// TIA Portal V16 export
// export: Created 2025-10-07T21:39:07.5159654Z, ExportSetting WithDefaults, DisplayName Totally Integrated Automation Portal, DisplayVersion V16, DisplayName TIA Portal Version Control Interface, DisplayVersion V16, DisplayName TIA Portal Openness, DisplayVersion V16, DisplayName STEP 7 Professional, DisplayVersion V16, DisplayName STEP 7 Safety, DisplayVersion V16, DisplayName WinCC Advanced, DisplayVersion V16
FUNCTION "5 - Prog. 3" : Void   // FC3, LAD
TITLE = System Program 3
VERSION : 0.1
// stored: AutoNumber true, IsIECCheckEnabled false, UDAEnableTagReadback false
   VAR_TEMP
      BlowOffTimer : Bool;
      Democoil : Bool;
      StartBlowOff : Bool;
      Pos2_Done : Bool;
      BlowOff_Activated : Bool;
      Retourband_Delayed : Bool;
      AandrukCilindersOut : Bool;
      Move2Busy : Bool;
      ProductBehindWals : Bool;
      SR_Move2 : Bool;
      Move1Busy : Bool;
   END_VAR
   VAR_TEMP   // added for the SCL form of the ladder/FBD networks
      _w1 : Bool;
   END_VAR
BEGIN

REGION Network 1: Close 1 Magazine Hole (cilinder)
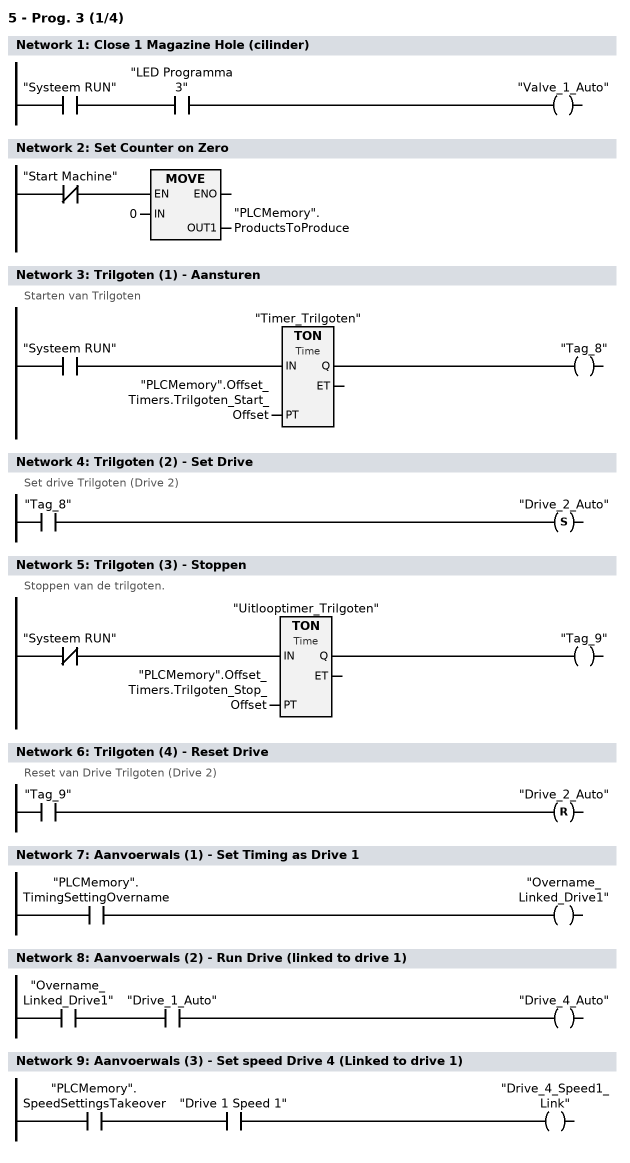
   RUNG wire#powerrail
      Contact( "Systeem RUN" )
      Contact( "LED Programma 3" )
      Coil( "Valve_1_Auto" )
   END_RUNG
   // the same network as SCL:
   "Valve_1_Auto" := "Systeem RUN" AND "LED Programma 3";
END_REGION

REGION Network 2: Set Counter on Zero
   RUNG wire#powerrail
      I_Contact( "Start Machine" )
      { S7_GenerateENO := "TRUE" } Move(in := 0, out1 => "PLCMemory".ProductsToProduce)
   END_RUNG
   // the same network as SCL:
   IF NOT "Start Machine" THEN "PLCMemory".ProductsToProduce := 0; END_IF;
END_REGION

REGION Network 3: Trilgoten (1) - Aansturen
   // Starten van Trilgoten
   RUNG wire#powerrail
      Contact( "Systeem RUN" )
      { S7_Templates := "time_type := Time" } "Timer_Trilgoten".TON(pt := "PLCMemory".Offset_Timers.Trilgoten_Start_Offset, et =>)
      Coil( "Tag_8" )
   END_RUNG
   // the same network as SCL:
   "Timer_Trilgoten".TON(IN := "Systeem RUN", PT := "PLCMemory".Offset_Timers.Trilgoten_Start_Offset);
   "Tag_8" := "Timer_Trilgoten".Q;
END_REGION

REGION Network 4: Trilgoten (2) - Set Drive
   // Set drive Trilgoten (Drive 2)
   RUNG wire#powerrail
      Contact( "Tag_8" )
      S_Coil( "Drive_2_Auto" )
   END_RUNG
   // the same network as SCL:
   IF "Tag_8" THEN "Drive_2_Auto" := TRUE; END_IF;
END_REGION

REGION Network 5: Trilgoten (3) - Stoppen
   // Stoppen van de trilgoten.
   RUNG wire#powerrail
      I_Contact( "Systeem RUN" )
      { S7_Templates := "time_type := Time" } "Uitlooptimer_Trilgoten".TON(pt := "PLCMemory".Offset_Timers.Trilgoten_Stop_Offset, et =>)
      Coil( "Tag_9" )
   END_RUNG
   // the same network as SCL:
   "Uitlooptimer_Trilgoten".TON(IN := NOT "Systeem RUN", PT := "PLCMemory".Offset_Timers.Trilgoten_Stop_Offset);
   "Tag_9" := "Uitlooptimer_Trilgoten".Q;
END_REGION

REGION Network 6: Trilgoten (4) - Reset Drive
   // Reset van Drive Trilgoten (Drive 2)
   RUNG wire#powerrail
      Contact( "Tag_9" )
      R_Coil( "Drive_2_Auto" )
   END_RUNG
   // the same network as SCL:
   IF "Tag_9" THEN "Drive_2_Auto" := FALSE; END_IF;
END_REGION

REGION Network 7: Aanvoerwals (1) - Set Timing as Drive 1
   RUNG wire#powerrail
      Contact( "PLCMemory".TimingSettingOvername )
      Coil( "Overname_Linked_Drive1" )
   END_RUNG
   // the same network as SCL:
   "Overname_Linked_Drive1" := "PLCMemory".TimingSettingOvername;
END_REGION

REGION Network 8: Aanvoerwals (2) - Run Drive (linked to drive 1)
   RUNG wire#powerrail
      Contact( "Overname_Linked_Drive1" )
      Contact( "Drive_1_Auto" )
      Coil( "Drive_4_Auto" )
   END_RUNG
   // the same network as SCL:
   "Drive_4_Auto" := "Overname_Linked_Drive1" AND "Drive_1_Auto";
END_REGION

REGION Network 9: Aanvoerwals (3) - Set speed Drive 4 (Linked to drive 1)
   RUNG wire#powerrail
      Contact( "PLCMemory".SpeedSettingsTakeover )
      Contact( "Drive 1 Speed 1" )
      Coil( "Drive_4_Speed1_Link" )
   END_RUNG
   // the same network as SCL:
   "Drive_4_Speed1_Link" := "PLCMemory".SpeedSettingsTakeover AND "Drive 1 Speed 1";
END_REGION

REGION Network 10: Aanvoerwals (4) - Set alternative Speed 1
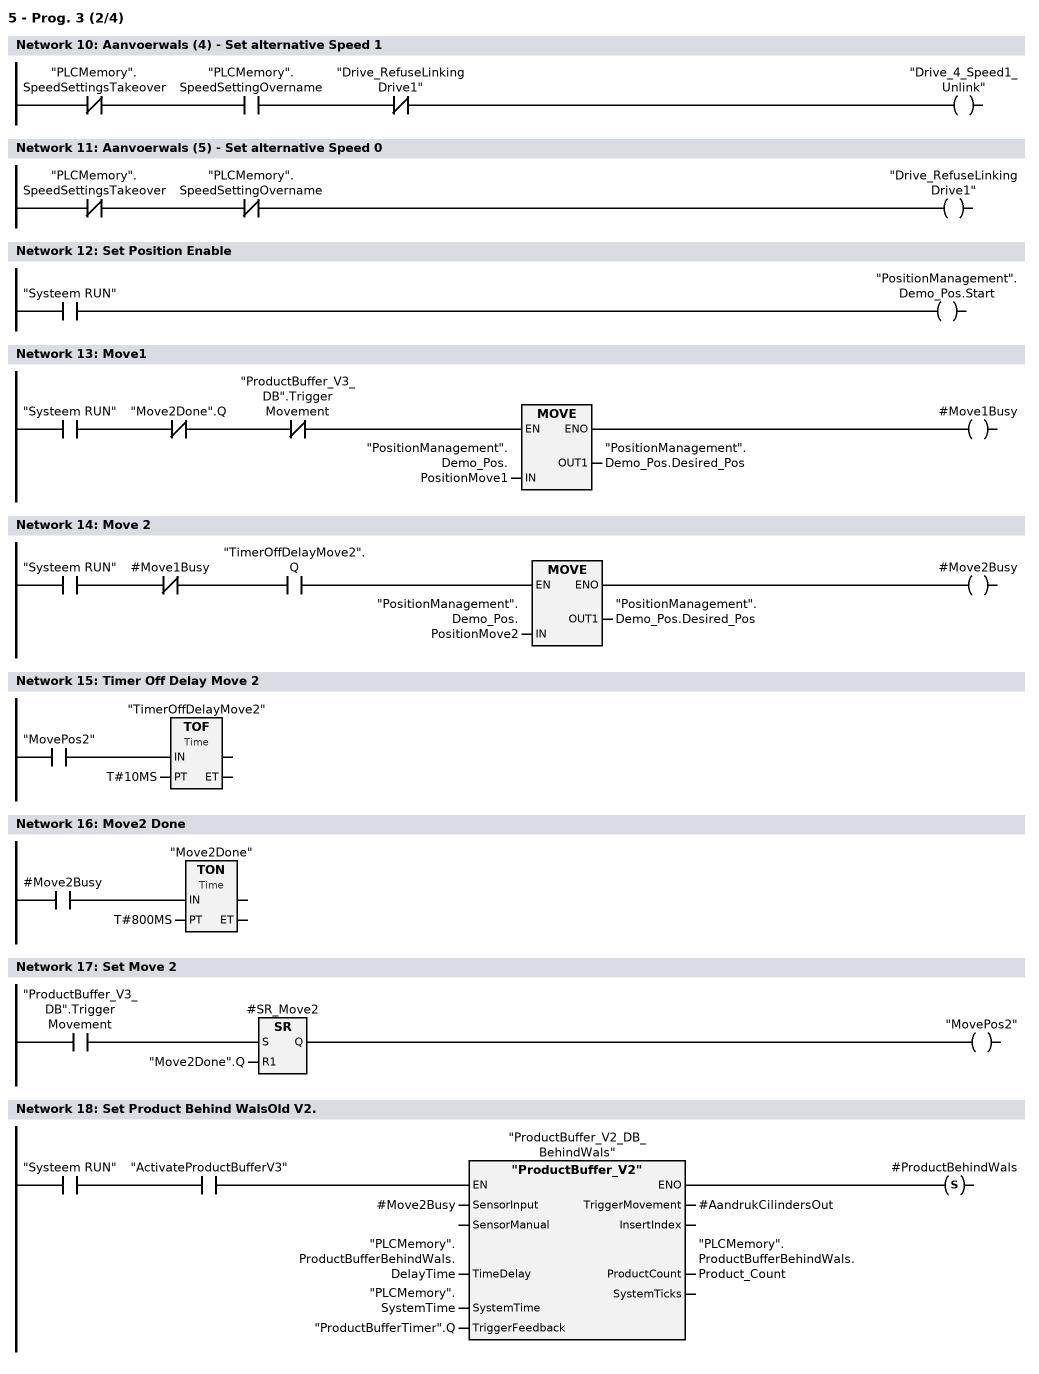
   RUNG wire#powerrail
      I_Contact( "PLCMemory".SpeedSettingsTakeover )
      Contact( "PLCMemory".SpeedSettingOvername )
      I_Contact( "Drive_RefuseLinkingDrive1" )
      Coil( "Drive_4_Speed1_Unlink" )
   END_RUNG
   // the same network as SCL:
   "Drive_4_Speed1_Unlink" := NOT "PLCMemory".SpeedSettingsTakeover AND "PLCMemory".SpeedSettingOvername AND NOT "Drive_RefuseLinkingDrive1";
END_REGION

REGION Network 11: Aanvoerwals (5) - Set alternative Speed 0
   RUNG wire#powerrail
      I_Contact( "PLCMemory".SpeedSettingsTakeover )
      I_Contact( "PLCMemory".SpeedSettingOvername )
      Coil( "Drive_RefuseLinkingDrive1" )
   END_RUNG
   // the same network as SCL:
   "Drive_RefuseLinkingDrive1" := NOT "PLCMemory".SpeedSettingsTakeover AND NOT "PLCMemory".SpeedSettingOvername;
END_REGION

REGION Network 12: Set Position Enable
   RUNG wire#powerrail
      Contact( "Systeem RUN" )
      Coil( "PositionManagement".Demo_Pos.Start )
   END_RUNG
   // the same network as SCL:
   "PositionManagement".Demo_Pos.Start := "Systeem RUN";
END_REGION

REGION Network 13: Move1
   RUNG wire#powerrail
      Contact( "Systeem RUN" )
      I_Contact( "Move2Done".Q )
      I_Contact( "ProductBuffer_V3_DB".TriggerMovement )
      { S7_GenerateENO := "TRUE" } Move(in := "PositionManagement".Demo_Pos.PositionMove1, out1 => "PositionManagement".Demo_Pos.Desired_Pos)
      Coil( #Move1Busy )
   END_RUNG
   // the same network as SCL:
   // ENO of a box is taken as its EN; it also drops when the box reports an error
   #_w1 := "Systeem RUN" AND NOT "Move2Done".Q AND NOT "ProductBuffer_V3_DB".TriggerMovement;
   IF #_w1 THEN
       "PositionManagement".Demo_Pos.Desired_Pos := "PositionManagement".Demo_Pos.PositionMove1;
   END_IF;
   #Move1Busy := #_w1;
END_REGION

REGION Network 14: Move 2
   RUNG wire#powerrail
      Contact( "Systeem RUN" )
      I_Contact( #Move1Busy )
      Contact( "TimerOffDelayMove2".Q )
      { S7_GenerateENO := "TRUE" } Move(in := "PositionManagement".Demo_Pos.PositionMove2, out1 => "PositionManagement".Demo_Pos.Desired_Pos)
      Coil( #Move2Busy )
   END_RUNG
   // the same network as SCL:
   // ENO of a box is taken as its EN; it also drops when the box reports an error
   #_w1 := "Systeem RUN" AND NOT #Move1Busy AND "TimerOffDelayMove2".Q;
   IF #_w1 THEN
       "PositionManagement".Demo_Pos.Desired_Pos := "PositionManagement".Demo_Pos.PositionMove2;
   END_IF;
   #Move2Busy := #_w1;
END_REGION

REGION Network 15: Timer Off Delay Move 2
   RUNG wire#powerrail
      Contact( "MovePos2" )
      { S7_Templates := "time_type := Time" } "TimerOffDelayMove2".TOF(pt := T#10MS, et =>)
   END_RUNG
   // the same network as SCL:
   "TimerOffDelayMove2".TOF(IN := "MovePos2", PT := T#10MS);
END_REGION

REGION Network 16: Move2 Done
   RUNG wire#powerrail
      Contact( #Move2Busy )
      { S7_Templates := "time_type := Time" } "Move2Done".TON(pt := T#800MS, et =>)
   END_RUNG
   // the same network as SCL:
   "Move2Done".TON(IN := #Move2Busy, PT := T#800MS);
END_REGION

REGION Network 17: Set Move 2
   RUNG wire#powerrail
      Contact( "ProductBuffer_V3_DB".TriggerMovement )
      S_SR(operand := #SR_Move2, r1 := "Move2Done".Q)
      Coil( "MovePos2" )
   END_RUNG
   // the same network as SCL:
   IF "ProductBuffer_V3_DB".TriggerMovement THEN
       #SR_Move2 := TRUE;   // SR flip-flop
   END_IF;
   IF "Move2Done".Q THEN #SR_Move2 := FALSE; END_IF;
   "MovePos2" := #SR_Move2;
END_REGION

REGION Network 18: Set Product Behind WalsOld V2.
   RUNG wire#powerrail
      Contact( "Systeem RUN" )
      Contact( "ActivateProductBufferV3" )
      "ProductBuffer_V2_DB_BehindWals"(SensorInput := #Move2Busy, SensorManual :=, TimeDelay := "PLCMemory".ProductBufferBehindWals.DelayTime, SystemTime := "PLCMemory".SystemTime, TriggerFeedback := "ProductBufferTimer".Q, TriggerMovement => #AandrukCilindersOut, InsertIndex =>, ProductCount => "PLCMemory".ProductBufferBehindWals.Product_Count, SystemTicks =>)
      S_Coil( #ProductBehindWals )
   END_RUNG
   // the same network as SCL:
   "ProductBuffer_V2_DB_BehindWals"(EN := "Systeem RUN" AND "ActivateProductBufferV3",   // "ProductBuffer_V2"
                           SensorInput := #Move2Busy,
                           TimeDelay := "PLCMemory".ProductBufferBehindWals.DelayTime,
                           SystemTime := "PLCMemory".SystemTime,
                           TriggerFeedback := "ProductBufferTimer".Q,
                           TriggerMovement => #AandrukCilindersOut,
                           ProductCount => "PLCMemory".ProductBufferBehindWals.Product_Count,
                           ENO => #_w1);
   IF #_w1 THEN #ProductBehindWals := TRUE; END_IF;
END_REGION

REGION Network 19: PorductBuffer Behind Wals V3
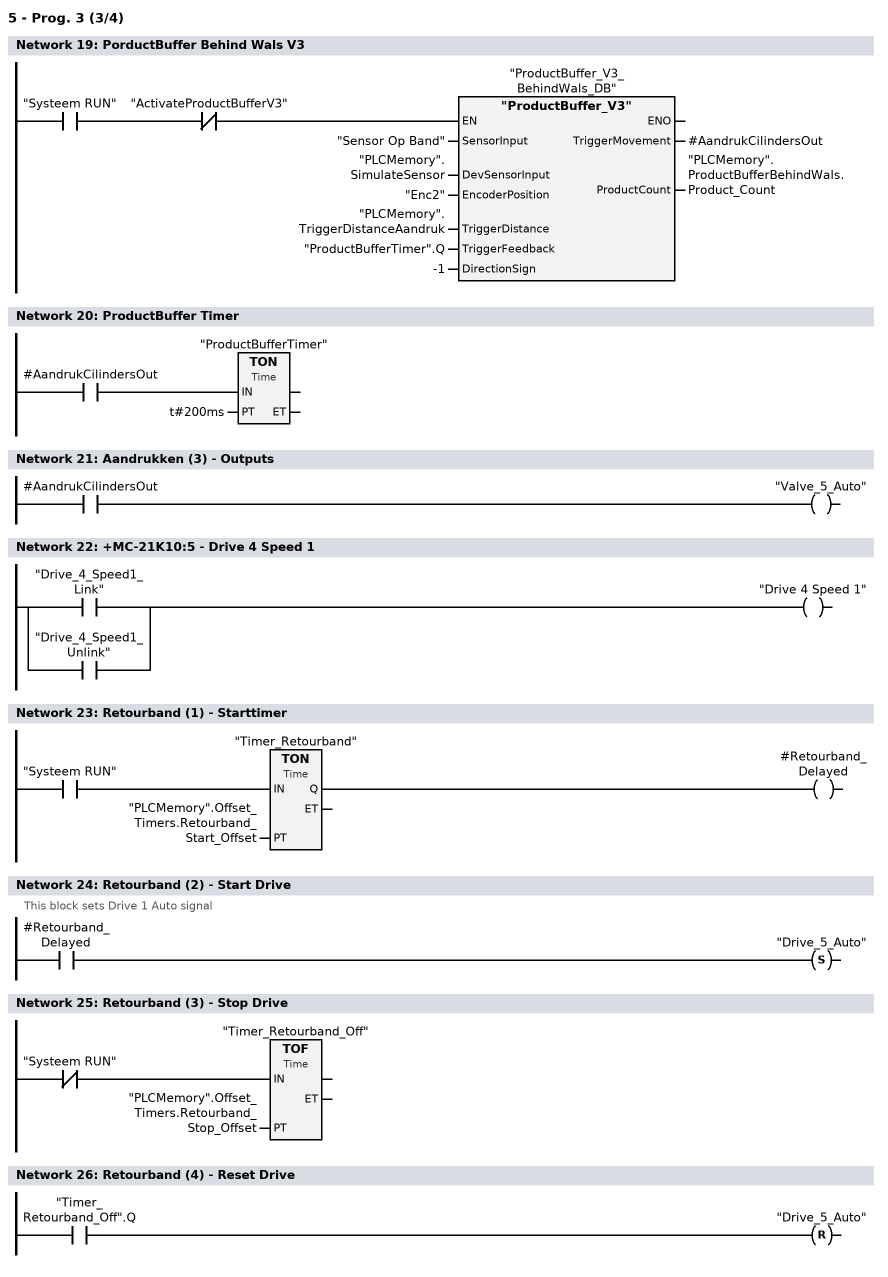
   RUNG wire#powerrail
      Contact( "Systeem RUN" )
      I_Contact( "ActivateProductBufferV3" )
      "ProductBuffer_V3_BehindWals_DB"(SensorInput := "Sensor Op Band", DevSensorInput := "PLCMemory".SimulateSensor, EncoderPosition := "Enc2", TriggerDistance := "PLCMemory".TriggerDistanceAandruk, TriggerFeedback := "ProductBufferTimer".Q, DirectionSign := -1, TriggerMovement => #AandrukCilindersOut, ProductCount => "PLCMemory".ProductBufferBehindWals.Product_Count)
   END_RUNG
   // the same network as SCL:
   IF "Systeem RUN" AND NOT "ActivateProductBufferV3" THEN
       "ProductBuffer_V3_BehindWals_DB"(SensorInput := "Sensor Op Band",   // "ProductBuffer_V3"
                               DevSensorInput := "PLCMemory".SimulateSensor,
                               EncoderPosition := "Enc2",
                               TriggerDistance := "PLCMemory".TriggerDistanceAandruk,
                               TriggerFeedback := "ProductBufferTimer".Q,
                               DirectionSign := -1,
                               TriggerMovement => #AandrukCilindersOut,
                               ProductCount => "PLCMemory".ProductBufferBehindWals.Product_Count);
   END_IF;
END_REGION

REGION Network 20: ProductBuffer Timer
   RUNG wire#powerrail
      Contact( #AandrukCilindersOut )
      { S7_Templates := "time_type := Time" } "ProductBufferTimer".TON(pt := t#200ms, et =>)
   END_RUNG
   // the same network as SCL:
   "ProductBufferTimer".TON(IN := #AandrukCilindersOut, PT := t#200ms);
END_REGION

REGION Network 21: Aandrukken (3) - Outputs
   RUNG wire#powerrail
      Contact( #AandrukCilindersOut )
      Coil( "Valve_5_Auto" )
   END_RUNG
   // the same network as SCL:
   "Valve_5_Auto" := #AandrukCilindersOut;
END_REGION

REGION Network 22: +MC-21K10:5 - Drive 4 Speed 1
   RUNG wire#powerrail
      Contact( "Drive_4_Speed1_Link" )
      wire#w1
      Coil( "Drive 4 Speed 1" )
   END_RUNG
   RUNG wire#powerrail
      Contact( "Drive_4_Speed1_Unlink" )
   END_RUNG wire#w1
   // the same network as SCL:
   "Drive 4 Speed 1" := "Drive_4_Speed1_Link" OR "Drive_4_Speed1_Unlink";
END_REGION

REGION Network 23: Retourband (1) - Starttimer
   RUNG wire#powerrail
      Contact( "Systeem RUN" )
      { S7_Templates := "time_type := Time" } "Timer_Retourband".TON(pt := "PLCMemory".Offset_Timers.Retourband_Start_Offset, et =>)
      Coil( #Retourband_Delayed )
   END_RUNG
   // the same network as SCL:
   "Timer_Retourband".TON(IN := "Systeem RUN", PT := "PLCMemory".Offset_Timers.Retourband_Start_Offset);
   #Retourband_Delayed := "Timer_Retourband".Q;
END_REGION

REGION Network 24: Retourband (2) - Start Drive
   // This block sets Drive 1 Auto signal
   RUNG wire#powerrail
      Contact( #Retourband_Delayed )
      S_Coil( "Drive_5_Auto" )
   END_RUNG
   // the same network as SCL:
   IF #Retourband_Delayed THEN "Drive_5_Auto" := TRUE; END_IF;
END_REGION

REGION Network 25: Retourband (3) - Stop Drive
   RUNG wire#powerrail
      I_Contact( "Systeem RUN" )
      { S7_Templates := "time_type := Time" } "Timer_Retourband_Off".TOF(pt := "PLCMemory".Offset_Timers.Retourband_Stop_Offset, et =>)
   END_RUNG
   // the same network as SCL:
   "Timer_Retourband_Off".TOF(IN := NOT "Systeem RUN", PT := "PLCMemory".Offset_Timers.Retourband_Stop_Offset);
END_REGION

REGION Network 26: Retourband (4) - Reset Drive
   RUNG wire#powerrail
      Contact( "Timer_Retourband_Off".Q )
      R_Coil( "Drive_5_Auto" )
   END_RUNG
   // the same network as SCL:
   IF "Timer_Retourband_Off".Q THEN "Drive_5_Auto" := FALSE; END_IF;
END_REGION

REGION Network 27: Blow off (1) - Set Blow Off Timer
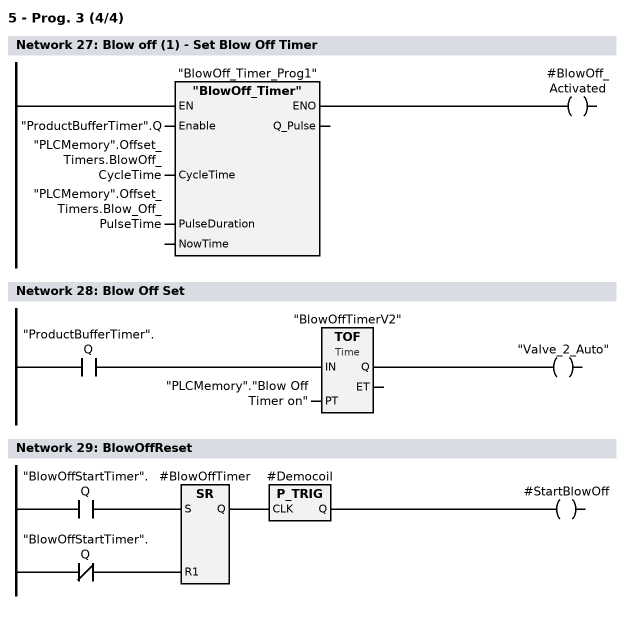
   RUNG wire#powerrail
      "BlowOff_Timer_Prog1"(Enable := "ProductBufferTimer".Q, CycleTime := "PLCMemory".Offset_Timers.BlowOff_CycleTime, PulseDuration := "PLCMemory".Offset_Timers.Blow_Off_PulseTime, NowTime :=, Q_Pulse =>)
      Coil( #BlowOff_Activated )
   END_RUNG
   // the same network as SCL:
   "BlowOff_Timer_Prog1"(Enable := "ProductBufferTimer".Q,   // "BlowOff_Timer"
                         CycleTime := "PLCMemory".Offset_Timers.BlowOff_CycleTime,
                         PulseDuration := "PLCMemory".Offset_Timers.Blow_Off_PulseTime,
                         ENO => #_w1);
   #BlowOff_Activated := #_w1;
END_REGION

REGION Network 28: Blow Off Set
   RUNG wire#powerrail
      Contact( "ProductBufferTimer".Q )
      { S7_Templates := "time_type := Time" } "BlowOffTimerV2".TOF(pt := "PLCMemory"."Blow Off Timer on", et =>)
      Coil( "Valve_2_Auto" )
   END_RUNG
   // the same network as SCL:
   "BlowOffTimerV2".TOF(IN := "ProductBufferTimer".Q, PT := "PLCMemory"."Blow Off Timer on");
   "Valve_2_Auto" := "BlowOffTimerV2".Q;
END_REGION

REGION Network 29: BlowOffReset
   RUNG wire#powerrail
      Contact( "BlowOffStartTimer".Q )
      S_SR(operand := #BlowOffTimer, r1 := wire#w1)
      P_Trig( #Democoil )
      Coil( #StartBlowOff )
   END_RUNG
   RUNG wire#powerrail
      I_Contact( "BlowOffStartTimer".Q )
   END_RUNG wire#w1
   // the same network as SCL:
   IF "BlowOffStartTimer".Q THEN
       #BlowOffTimer := TRUE;   // SR flip-flop
   END_IF;
   IF NOT "BlowOffStartTimer".Q THEN #BlowOffTimer := FALSE; END_IF;
   #_w1 := #BlowOffTimer AND NOT #Democoil;   // rising edge
   #Democoil := #BlowOffTimer;
   #StartBlowOff := #_w1;
END_REGION
END_FUNCTION
